Staubli VAL3: vec2num.pgx

public program vec2num(string& x_sInput[], num& x_nResult[])
  local num l_nLength
  local num l_nElement
  local string l_sCopy
  local num l_nValue
  local bool l_bSucces
  local num l_nSucessCounter
begin

  l_nLength = size(x_sInput)
  x_nResult[0] = 0
  resize(x_nResult,1,1)

  for l_nElement = 0 to l_nLength-1
    // copy element
    l_sCopy = x_sInput[l_nElement]
    toNum(l_sCopy, l_nValue, l_bSucces)
    if l_bSucces
      if l_nElement !=0
        append(x_nResult)
      endIf
      x_nResult[l_nSucessCounter] = l_nValue
      l_nSucessCounter = l_nSucessCounter +1
    endIf
  endFor

end
